Yaskawa INFORM job: plaster_roller_planes_program.JBI

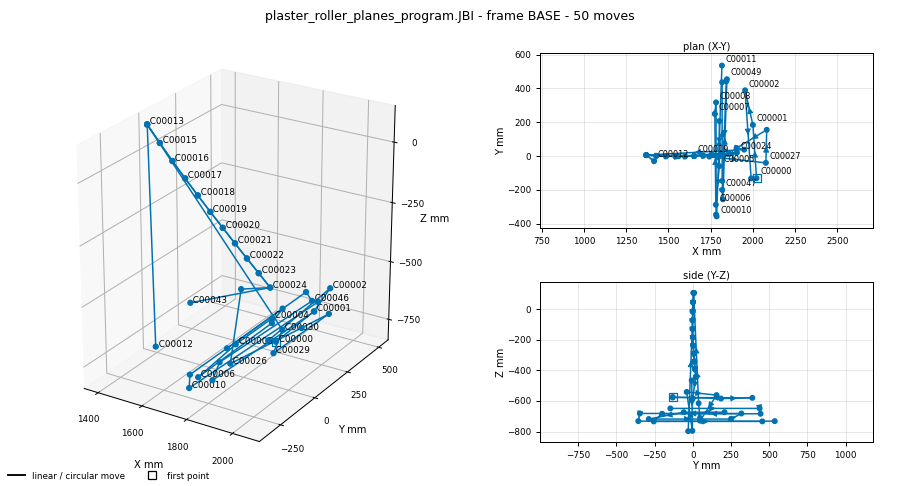
[picture p0: tool path of plaster_roller_planes_program.JBI in frame BASE, 50 of 55 moves have a stored position in this frame; points joined in program order, loops and branches not executed]
/JOB
//NAME plaster_roller_planes_program
//POS
///NPOS 50,0,50,0,0,0
///TOOL 0
///POSTYPE BASE
///RECTAN
///RCONF 0,0,0,0,0,0,0,0,0,0,0,0,0,0,0,0,0,0,0,0,0,0,0,0
C00000=2021.234573,-131.092234,-574.555100,175.000000,-5.000000,5.000000
C00001=1999.638324,184.290315,-584.470091,175.000000,-5.000000,5.000000
C00002=1953.430568,389.362677,-579.865091,175.000000,-5.000000,5.000000
C00003=1989.138795,-132.105268,-577.415091,175.000000,-5.000000,5.000000
C00004=1800.999949,207.228223,-673.785781,-175.000000,-89.477998,5.000000
C00005=1801.035871,-59.250538,-673.803283,-175.000000,-89.477998,5.000000
C00006=1780.197968,-288.172557,-718.609235,-175.000000,-89.477998,5.000000
C00007=1774.331989,249.242822,-718.521157,-175.000000,-89.477998,5.000000
C00008=1781.677406,317.567157,-681.983209,-175.000000,-89.477998,5.000000
C00009=1781.712974,-346.269616,-682.026316,-175.000000,-89.477998,5.000000
C00010=1784.916975,-356.713030,-732.058254,-175.000000,-89.477998,5.000000
C00011=1816.442815,535.742557,-732.287952,180.000000,-60.000000,0.000000
C00012=1414.870786,-30.200631,-797.980210,175.000000,-44.008636,5.000000
C00013=1368.810726,5.598725,106.220809,10.334919,12.478409,-175.000000
C00014=1368.722137,5.635807,106.210519,10.335309,12.479805,-175.000000
C00015=1427.664073,1.310744,45.164513,8.007028,15.446309,-175.000000
C00016=1485.342476,-1.169304,-14.461285,5.836768,18.504360,-175.000000
C00017=1542.137536,-2.013853,-72.457017,5.000000,21.645330,-175.000000
C00018=1597.803707,-1.547920,-129.272262,5.000000,24.851409,-175.000000
C00019=1652.131552,0.101403,-184.539036,5.000000,28.105997,-175.000000
C00020=1705.342433,2.685647,-238.323026,5.000000,-31.424829,5.000000
C00021=1757.041585,6.061019,-291.005597,-5.000000,-34.810443,5.000000
C00022=1807.502837,10.194566,-342.680585,5.000000,-38.223195,5.000000
C00023=1856.514365,14.798073,-393.087178,-5.000000,-41.626153,5.000000
C00024=1903.964863,19.981849,-442.804263,-5.000000,-44.999700,5.000000
C00025=1792.718634,-7.244186,-466.143732,175.000000,5.000000,5.000000
C00026=1741.464877,-3.097369,-795.911117,174.314304,22.844892,-5.000000
C00027=2076.479855,-40.177964,-541.339182,-157.727499,15.081099,6.082723
C00028=2081.465579,155.420071,-562.072620,149.632165,15.624200,-8.967879
C00029=1903.620197,47.525247,-729.388818,-174.607663,21.860553,5.000000
C00030=1947.795433,37.964353,-615.310732,175.000000,5.000000,5.000000
C00031=1368.810726,5.598725,106.220809,10.334919,12.478409,-175.000000
C00032=1368.722137,5.635807,106.210519,10.335309,12.479805,-175.000000
C00033=1427.664073,1.310744,45.164513,8.007028,15.446309,-175.000000
C00034=1485.342476,-1.169304,-14.461285,5.836768,18.504360,-175.000000
C00035=1542.137536,-2.013853,-72.457017,5.000000,21.645330,-175.000000
C00036=1597.803707,-1.547920,-129.272262,5.000000,24.851409,-175.000000
C00037=1652.131552,0.101403,-184.539036,5.000000,28.105997,-175.000000
C00038=1705.342433,2.685647,-238.323026,5.000000,-31.424829,5.000000
C00039=1757.041585,6.061019,-291.005597,-5.000000,-34.810443,5.000000
C00040=1807.502837,10.194566,-342.680585,5.000000,-38.223195,5.000000
C00041=1856.514365,14.798073,-393.087178,-5.000000,-41.626153,5.000000
C00042=1903.964863,19.981849,-442.804263,-5.000000,-44.999700,5.000000
C00043=1559.432639,-1.164519,-584.123732,180.000000,-60.000000,0.000000
C00044=1817.897487,-146.789716,-648.928907,5.000000,-89.672961,-175.000000
C00045=1817.529013,436.965166,-648.945923,5.000000,-89.672961,-175.000000
C00046=1842.122086,442.917509,-683.999202,5.000000,-89.672961,-175.000000
C00047=1818.222269,-199.903953,-684.119208,5.000000,-89.672961,-175.000000
C00048=1821.926379,-255.543191,-734.097457,5.000000,-89.672961,-175.000000
C00049=1846.110777,454.677474,-733.977549,180.000000,-60.000000,0.000000
///POSTYPE PULSE
///PULSE
EC00000=4096.0
EC00001=4096.0
EC00002=4096.0
EC00003=4096.0
EC00004=183296.0
EC00005=183296.0
EC00006=183296.0
EC00007=183296.0
EC00008=183296.0
EC00009=183296.0
EC00010=183296.0
EC00011=183296.0
EC00012=282624.0
EC00013=282624.0
EC00014=282624.0
EC00015=282624.0
EC00016=282624.0
EC00017=282624.0
EC00018=282624.0
EC00019=282624.0
EC00020=282624.0
EC00021=282624.0
EC00022=282624.0
EC00023=282624.0
EC00024=282624.0
EC00025=282624.0
EC00026=282624.0
EC00027=282624.0
EC00028=282624.0
EC00029=282624.0
EC00030=282624.0
EC00031=282624.0
EC00032=282624.0
EC00033=282624.0
EC00034=282624.0
EC00035=282624.0
EC00036=282624.0
EC00037=282624.0
EC00038=282624.0
EC00039=282624.0
EC00040=282624.0
EC00041=282624.0
EC00042=282624.0
EC00043=282624.0
EC00044=367616.0
EC00045=367616.0
EC00046=367616.0
EC00047=367616.0
EC00048=367616.0
EC00049=367616.0
//INST
///DATE 2023/08/16 17:22
///ATTR SC,RW,RJ
////FRAME BASE
///GROUP1 RB1,ST1
NOP
MOVJ P009 EX000 VJ=15.00
MOVJ C00000 EC00000 VJ=15.0
CALL JOB:SPYON
MOVL C00001 EC00001 V=150.0
MOVL C00002 EC00002 V=150.0
MOVL C00003 EC00003 V=150.0
CALL JOB:SPYOF
MOVJ P009 VJ=15.00
MOVJ C00004 EC00004 VJ=15.0
CALL JOB:SPYON
MOVL C00005 EC00005 V=150.0
MOVL C00006 EC00006 V=150.0
MOVL C00007 EC00007 V=150.0
MOVL C00008 EC00008 V=150.0
MOVL C00009 EC00009 V=150.0
MOVL C00010 EC00010 V=150.0
MOVL C00011 EC00011 V=150.0
CALL JOB:SPYOF
MOVJ P009 VJ=15.00
MOVJ C00012 EC00012 VJ=15.0
CALL JOB:SPYON
MOVL C00013 EC00013 V=150.0
MOVL C00014 EC00014 V=150.0
MOVL C00015 EC00015 V=150.0
MOVL C00016 EC00016 V=150.0
MOVL C00017 EC00017 V=150.0
MOVL C00018 EC00018 V=150.0
MOVL C00019 EC00019 V=150.0
MOVL C00020 EC00020 V=150.0
MOVL C00021 EC00021 V=150.0
MOVL C00022 EC00022 V=150.0
MOVL C00023 EC00023 V=150.0
MOVL C00024 EC00024 V=150.0
MOVL C00025 EC00025 V=150.0
MOVL C00026 EC00026 V=150.0
MOVL C00027 EC00027 V=150.0
MOVL C00028 EC00028 V=150.0
MOVL C00029 EC00029 V=150.0
MOVL C00030 EC00030 V=150.0
MOVL C00031 EC00031 V=150.0
MOVL C00032 EC00032 V=150.0
MOVL C00033 EC00033 V=150.0
MOVL C00034 EC00034 V=150.0
MOVL C00035 EC00035 V=150.0
MOVL C00036 EC00036 V=150.0
MOVL C00037 EC00037 V=150.0
MOVL C00038 EC00038 V=150.0
MOVL C00039 EC00039 V=150.0
MOVL C00040 EC00040 V=150.0
MOVL C00041 EC00041 V=150.0
MOVL C00042 EC00042 V=150.0
MOVL C00043 EC00043 V=150.0
CALL JOB:SPYOF
MOVJ P009 VJ=15.00
MOVJ C00044 EC00044 VJ=15.0
CALL JOB:SPYON
MOVL C00045 EC00045 V=150.0
MOVL C00046 EC00046 V=150.0
MOVL C00047 EC00047 V=150.0
MOVL C00048 EC00048 V=150.0
MOVL C00049 EC00049 V=150.0
CALL JOB:SPYOF
MOVJ P009 VJ=15.00
END
